// TIA Portal V20 export
FUNCTION "CollectAlarms" : Void   // FC35, LAD
TITLE = U1Em5_CathodeMainPnP
// stored: Namespace Unit1.Em5, SetENOAutomatically false
   VAR_INPUT
      resetAlarms : Bool;
      disableAlarms : Bool;
   END_VAR
   VAR_OUTPUT
      commandsToUnit : "LUC_typeStateCommands";   // Feedback to the unit
   END_VAR
   VAR CONSTANT
      DelayTime : Time := T#300ms;
      NoDelayTime : Time;
   END_VAR
BEGIN

REGION Network 1: Reset Alarms
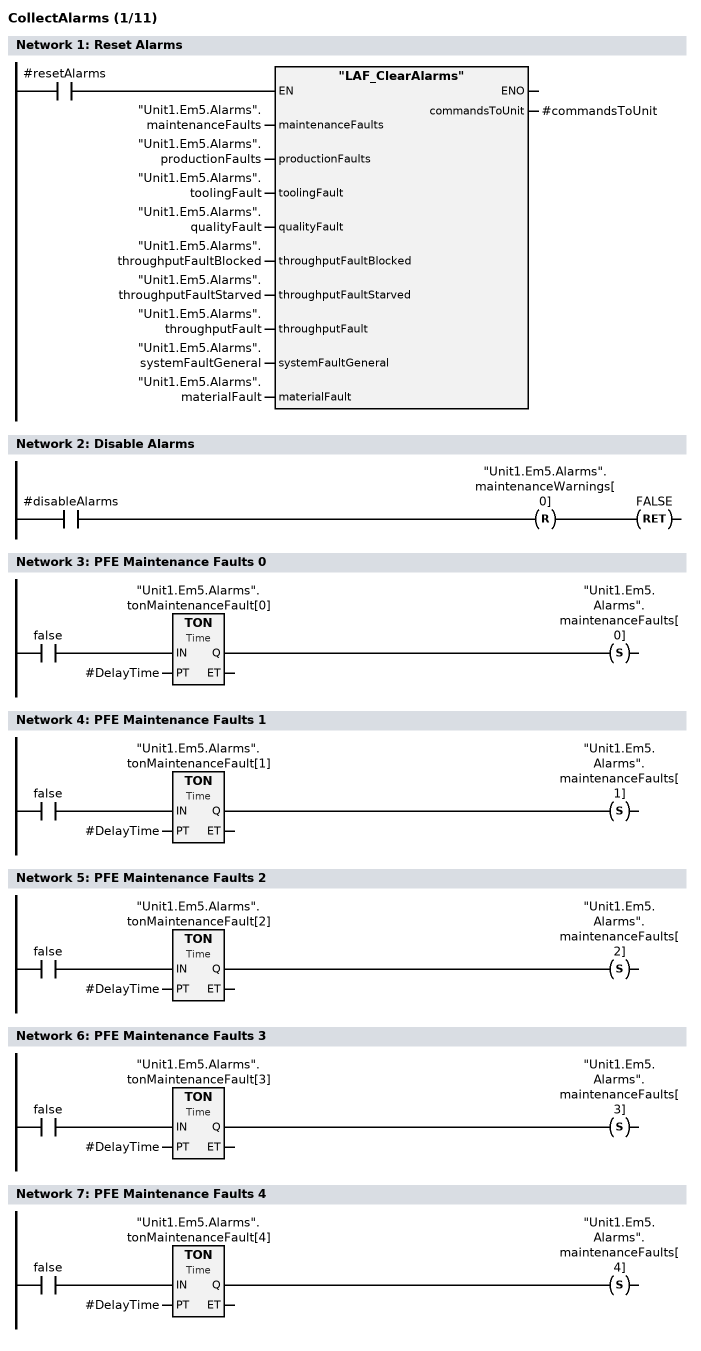
   RUNG wire#powerrail
      Contact( #resetAlarms )
      "LAF_ClearAlarms"(maintenanceFaults := "Unit1.Em5.Alarms".maintenanceFaults, productionFaults := "Unit1.Em5.Alarms".productionFaults, toolingFault := "Unit1.Em5.Alarms".toolingFault, qualityFault := "Unit1.Em5.Alarms".qualityFault, throughputFaultBlocked := "Unit1.Em5.Alarms".throughputFaultBlocked, throughputFaultStarved := "Unit1.Em5.Alarms".throughputFaultStarved, throughputFault := "Unit1.Em5.Alarms".throughputFault, systemFaultGeneral := "Unit1.Em5.Alarms".systemFaultGeneral, materialFault := "Unit1.Em5.Alarms".materialFault, commandsToUnit => #commandsToUnit)
   END_RUNG
   // the same network as SCL:
   IF #resetAlarms THEN
       "LAF_ClearAlarms"(maintenanceFaults := "Unit1.Em5.Alarms".maintenanceFaults,
                         productionFaults := "Unit1.Em5.Alarms".productionFaults,
                         toolingFault := "Unit1.Em5.Alarms".toolingFault,
                         qualityFault := "Unit1.Em5.Alarms".qualityFault,
                         throughputFaultBlocked := "Unit1.Em5.Alarms".throughputFaultBlocked,
                         throughputFaultStarved := "Unit1.Em5.Alarms".throughputFaultStarved,
                         throughputFault := "Unit1.Em5.Alarms".throughputFault,
                         systemFaultGeneral := "Unit1.Em5.Alarms".systemFaultGeneral,
                         materialFault := "Unit1.Em5.Alarms".materialFault,
                         commandsToUnit => #commandsToUnit);
   END_IF;
END_REGION

REGION Network 2: Disable Alarms
   RUNG wire#powerrail
      Contact( #disableAlarms )
      R_Coil( "Unit1.Em5.Alarms".maintenanceWarnings[0] )
      ReturnCoil( FALSE )
   END_RUNG
   // the same network as SCL:
   IF #disableAlarms THEN
       "Unit1.Em5.Alarms".maintenanceWarnings[0] := FALSE;
       ENO := FALSE;
       RETURN;
   END_IF;
END_REGION

REGION Network 3: PFE Maintenance Faults 0
   RUNG wire#powerrail
      Contact( false )
      { S7_Templates := "time_type := Time" } "Unit1.Em5.Alarms".tonMaintenanceFault[0].TON(pt := #DelayTime, et =>)
      S_Coil( "Unit1.Em5.Alarms".maintenanceFaults[0] )
   END_RUNG
   // the same network as SCL:
   "Unit1.Em5.Alarms".tonMaintenanceFault[0].TON(IN := false, PT := #DelayTime);
   IF "Unit1.Em5.Alarms".tonMaintenanceFault[0].Q THEN
       "Unit1.Em5.Alarms".maintenanceFaults[0] := TRUE;
   END_IF;
END_REGION

REGION Network 4: PFE Maintenance Faults 1
   RUNG wire#powerrail
      Contact( false )
      { S7_Templates := "time_type := Time" } "Unit1.Em5.Alarms".tonMaintenanceFault[1].TON(pt := #DelayTime, et =>)
      S_Coil( "Unit1.Em5.Alarms".maintenanceFaults[1] )
   END_RUNG
   // the same network as SCL:
   "Unit1.Em5.Alarms".tonMaintenanceFault[1].TON(IN := false, PT := #DelayTime);
   IF "Unit1.Em5.Alarms".tonMaintenanceFault[1].Q THEN
       "Unit1.Em5.Alarms".maintenanceFaults[1] := TRUE;
   END_IF;
END_REGION

REGION Network 5: PFE Maintenance Faults 2
   RUNG wire#powerrail
      Contact( false )
      { S7_Templates := "time_type := Time" } "Unit1.Em5.Alarms".tonMaintenanceFault[2].TON(pt := #DelayTime, et =>)
      S_Coil( "Unit1.Em5.Alarms".maintenanceFaults[2] )
   END_RUNG
   // the same network as SCL:
   "Unit1.Em5.Alarms".tonMaintenanceFault[2].TON(IN := false, PT := #DelayTime);
   IF "Unit1.Em5.Alarms".tonMaintenanceFault[2].Q THEN
       "Unit1.Em5.Alarms".maintenanceFaults[2] := TRUE;
   END_IF;
END_REGION

REGION Network 6: PFE Maintenance Faults 3
   RUNG wire#powerrail
      Contact( false )
      { S7_Templates := "time_type := Time" } "Unit1.Em5.Alarms".tonMaintenanceFault[3].TON(pt := #DelayTime, et =>)
      S_Coil( "Unit1.Em5.Alarms".maintenanceFaults[3] )
   END_RUNG
   // the same network as SCL:
   "Unit1.Em5.Alarms".tonMaintenanceFault[3].TON(IN := false, PT := #DelayTime);
   IF "Unit1.Em5.Alarms".tonMaintenanceFault[3].Q THEN
       "Unit1.Em5.Alarms".maintenanceFaults[3] := TRUE;
   END_IF;
END_REGION

REGION Network 7: PFE Maintenance Faults 4
   RUNG wire#powerrail
      Contact( false )
      { S7_Templates := "time_type := Time" } "Unit1.Em5.Alarms".tonMaintenanceFault[4].TON(pt := #DelayTime, et =>)
      S_Coil( "Unit1.Em5.Alarms".maintenanceFaults[4] )
   END_RUNG
   // the same network as SCL:
   "Unit1.Em5.Alarms".tonMaintenanceFault[4].TON(IN := false, PT := #DelayTime);
   IF "Unit1.Em5.Alarms".tonMaintenanceFault[4].Q THEN
       "Unit1.Em5.Alarms".maintenanceFaults[4] := TRUE;
   END_IF;
END_REGION

REGION Network 8: PFE Maintenance Faults 5
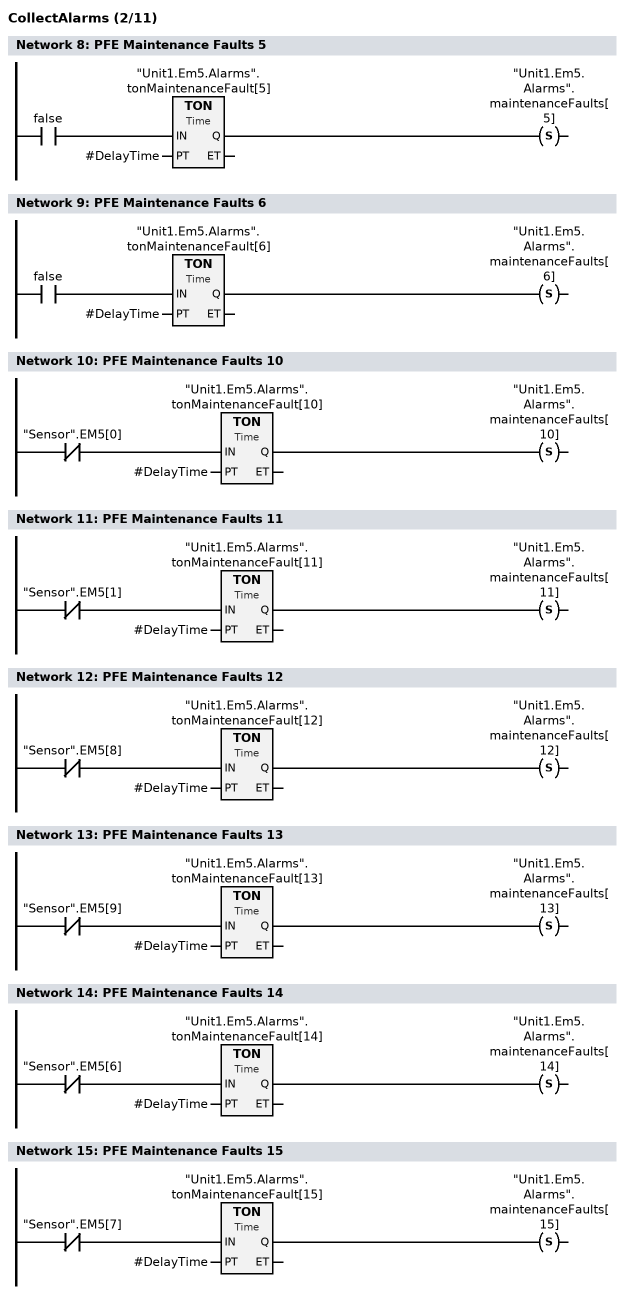
   RUNG wire#powerrail
      Contact( false )
      { S7_Templates := "time_type := Time" } "Unit1.Em5.Alarms".tonMaintenanceFault[5].TON(pt := #DelayTime, et =>)
      S_Coil( "Unit1.Em5.Alarms".maintenanceFaults[5] )
   END_RUNG
   // the same network as SCL:
   "Unit1.Em5.Alarms".tonMaintenanceFault[5].TON(IN := false, PT := #DelayTime);
   IF "Unit1.Em5.Alarms".tonMaintenanceFault[5].Q THEN
       "Unit1.Em5.Alarms".maintenanceFaults[5] := TRUE;
   END_IF;
END_REGION

REGION Network 9: PFE Maintenance Faults 6
   RUNG wire#powerrail
      Contact( false )
      { S7_Templates := "time_type := Time" } "Unit1.Em5.Alarms".tonMaintenanceFault[6].TON(pt := #DelayTime, et =>)
      S_Coil( "Unit1.Em5.Alarms".maintenanceFaults[6] )
   END_RUNG
   // the same network as SCL:
   "Unit1.Em5.Alarms".tonMaintenanceFault[6].TON(IN := false, PT := #DelayTime);
   IF "Unit1.Em5.Alarms".tonMaintenanceFault[6].Q THEN
       "Unit1.Em5.Alarms".maintenanceFaults[6] := TRUE;
   END_IF;
END_REGION

REGION Network 10: PFE Maintenance Faults 10
   RUNG wire#powerrail
      I_Contact( "Sensor".EM5[0] )
      { S7_Templates := "time_type := Time" } "Unit1.Em5.Alarms".tonMaintenanceFault[10].TON(pt := #DelayTime, et =>)
      S_Coil( "Unit1.Em5.Alarms".maintenanceFaults[10] )
   END_RUNG
   // the same network as SCL:
   "Unit1.Em5.Alarms".tonMaintenanceFault[10].TON(IN := NOT "Sensor".EM5[0], PT := #DelayTime);
   IF "Unit1.Em5.Alarms".tonMaintenanceFault[10].Q THEN
       "Unit1.Em5.Alarms".maintenanceFaults[10] := TRUE;
   END_IF;
END_REGION

REGION Network 11: PFE Maintenance Faults 11
   RUNG wire#powerrail
      I_Contact( "Sensor".EM5[1] )
      { S7_Templates := "time_type := Time" } "Unit1.Em5.Alarms".tonMaintenanceFault[11].TON(pt := #DelayTime, et =>)
      S_Coil( "Unit1.Em5.Alarms".maintenanceFaults[11] )
   END_RUNG
   // the same network as SCL:
   "Unit1.Em5.Alarms".tonMaintenanceFault[11].TON(IN := NOT "Sensor".EM5[1], PT := #DelayTime);
   IF "Unit1.Em5.Alarms".tonMaintenanceFault[11].Q THEN
       "Unit1.Em5.Alarms".maintenanceFaults[11] := TRUE;
   END_IF;
END_REGION

REGION Network 12: PFE Maintenance Faults 12
   RUNG wire#powerrail
      I_Contact( "Sensor".EM5[8] )
      { S7_Templates := "time_type := Time" } "Unit1.Em5.Alarms".tonMaintenanceFault[12].TON(pt := #DelayTime, et =>)
      S_Coil( "Unit1.Em5.Alarms".maintenanceFaults[12] )
   END_RUNG
   // the same network as SCL:
   "Unit1.Em5.Alarms".tonMaintenanceFault[12].TON(IN := NOT "Sensor".EM5[8], PT := #DelayTime);
   IF "Unit1.Em5.Alarms".tonMaintenanceFault[12].Q THEN
       "Unit1.Em5.Alarms".maintenanceFaults[12] := TRUE;
   END_IF;
END_REGION

REGION Network 13: PFE Maintenance Faults 13
   RUNG wire#powerrail
      I_Contact( "Sensor".EM5[9] )
      { S7_Templates := "time_type := Time" } "Unit1.Em5.Alarms".tonMaintenanceFault[13].TON(pt := #DelayTime, et =>)
      S_Coil( "Unit1.Em5.Alarms".maintenanceFaults[13] )
   END_RUNG
   // the same network as SCL:
   "Unit1.Em5.Alarms".tonMaintenanceFault[13].TON(IN := NOT "Sensor".EM5[9], PT := #DelayTime);
   IF "Unit1.Em5.Alarms".tonMaintenanceFault[13].Q THEN
       "Unit1.Em5.Alarms".maintenanceFaults[13] := TRUE;
   END_IF;
END_REGION

REGION Network 14: PFE Maintenance Faults 14
   RUNG wire#powerrail
      I_Contact( "Sensor".EM5[6] )
      { S7_Templates := "time_type := Time" } "Unit1.Em5.Alarms".tonMaintenanceFault[14].TON(pt := #DelayTime, et =>)
      S_Coil( "Unit1.Em5.Alarms".maintenanceFaults[14] )
   END_RUNG
   // the same network as SCL:
   "Unit1.Em5.Alarms".tonMaintenanceFault[14].TON(IN := NOT "Sensor".EM5[6], PT := #DelayTime);
   IF "Unit1.Em5.Alarms".tonMaintenanceFault[14].Q THEN
       "Unit1.Em5.Alarms".maintenanceFaults[14] := TRUE;
   END_IF;
END_REGION

REGION Network 15: PFE Maintenance Faults 15
   RUNG wire#powerrail
      I_Contact( "Sensor".EM5[7] )
      { S7_Templates := "time_type := Time" } "Unit1.Em5.Alarms".tonMaintenanceFault[15].TON(pt := #DelayTime, et =>)
      S_Coil( "Unit1.Em5.Alarms".maintenanceFaults[15] )
   END_RUNG
   // the same network as SCL:
   "Unit1.Em5.Alarms".tonMaintenanceFault[15].TON(IN := NOT "Sensor".EM5[7], PT := #DelayTime);
   IF "Unit1.Em5.Alarms".tonMaintenanceFault[15].Q THEN
       "Unit1.Em5.Alarms".maintenanceFaults[15] := TRUE;
   END_IF;
END_REGION

REGION Network 16: PFE Maintenance Faults 16
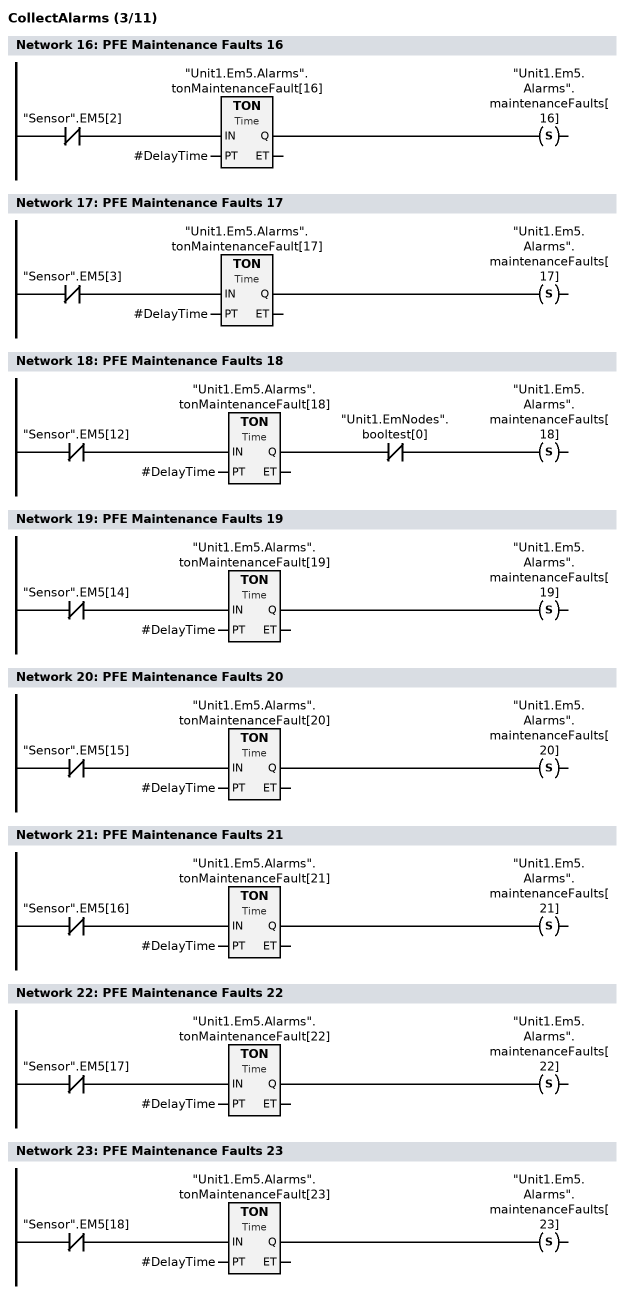
   RUNG wire#powerrail
      I_Contact( "Sensor".EM5[2] )
      { S7_Templates := "time_type := Time" } "Unit1.Em5.Alarms".tonMaintenanceFault[16].TON(pt := #DelayTime, et =>)
      S_Coil( "Unit1.Em5.Alarms".maintenanceFaults[16] )
   END_RUNG
   // the same network as SCL:
   "Unit1.Em5.Alarms".tonMaintenanceFault[16].TON(IN := NOT "Sensor".EM5[2], PT := #DelayTime);
   IF "Unit1.Em5.Alarms".tonMaintenanceFault[16].Q THEN
       "Unit1.Em5.Alarms".maintenanceFaults[16] := TRUE;
   END_IF;
END_REGION

REGION Network 17: PFE Maintenance Faults 17
   RUNG wire#powerrail
      I_Contact( "Sensor".EM5[3] )
      { S7_Templates := "time_type := Time" } "Unit1.Em5.Alarms".tonMaintenanceFault[17].TON(pt := #DelayTime, et =>)
      S_Coil( "Unit1.Em5.Alarms".maintenanceFaults[17] )
   END_RUNG
   // the same network as SCL:
   "Unit1.Em5.Alarms".tonMaintenanceFault[17].TON(IN := NOT "Sensor".EM5[3], PT := #DelayTime);
   IF "Unit1.Em5.Alarms".tonMaintenanceFault[17].Q THEN
       "Unit1.Em5.Alarms".maintenanceFaults[17] := TRUE;
   END_IF;
END_REGION

REGION Network 18: PFE Maintenance Faults 18
   RUNG wire#powerrail
      I_Contact( "Sensor".EM5[12] )
      { S7_Templates := "time_type := Time" } "Unit1.Em5.Alarms".tonMaintenanceFault[18].TON(pt := #DelayTime, et =>)
      I_Contact( "Unit1.EmNodes".booltest[0] )
      S_Coil( "Unit1.Em5.Alarms".maintenanceFaults[18] )
   END_RUNG
   // the same network as SCL:
   "Unit1.Em5.Alarms".tonMaintenanceFault[18].TON(IN := NOT "Sensor".EM5[12], PT := #DelayTime);
   IF "Unit1.Em5.Alarms".tonMaintenanceFault[18].Q AND NOT "Unit1.EmNodes".booltest[0] THEN
       "Unit1.Em5.Alarms".maintenanceFaults[18] := TRUE;
   END_IF;
END_REGION

REGION Network 19: PFE Maintenance Faults 19
   RUNG wire#powerrail
      I_Contact( "Sensor".EM5[14] )
      { S7_Templates := "time_type := Time" } "Unit1.Em5.Alarms".tonMaintenanceFault[19].TON(pt := #DelayTime, et =>)
      S_Coil( "Unit1.Em5.Alarms".maintenanceFaults[19] )
   END_RUNG
   // the same network as SCL:
   "Unit1.Em5.Alarms".tonMaintenanceFault[19].TON(IN := NOT "Sensor".EM5[14], PT := #DelayTime);
   IF "Unit1.Em5.Alarms".tonMaintenanceFault[19].Q THEN
       "Unit1.Em5.Alarms".maintenanceFaults[19] := TRUE;
   END_IF;
END_REGION

REGION Network 20: PFE Maintenance Faults 20
   RUNG wire#powerrail
      I_Contact( "Sensor".EM5[15] )
      { S7_Templates := "time_type := Time" } "Unit1.Em5.Alarms".tonMaintenanceFault[20].TON(pt := #DelayTime, et =>)
      S_Coil( "Unit1.Em5.Alarms".maintenanceFaults[20] )
   END_RUNG
   // the same network as SCL:
   "Unit1.Em5.Alarms".tonMaintenanceFault[20].TON(IN := NOT "Sensor".EM5[15], PT := #DelayTime);
   IF "Unit1.Em5.Alarms".tonMaintenanceFault[20].Q THEN
       "Unit1.Em5.Alarms".maintenanceFaults[20] := TRUE;
   END_IF;
END_REGION

REGION Network 21: PFE Maintenance Faults 21
   RUNG wire#powerrail
      I_Contact( "Sensor".EM5[16] )
      { S7_Templates := "time_type := Time" } "Unit1.Em5.Alarms".tonMaintenanceFault[21].TON(pt := #DelayTime, et =>)
      S_Coil( "Unit1.Em5.Alarms".maintenanceFaults[21] )
   END_RUNG
   // the same network as SCL:
   "Unit1.Em5.Alarms".tonMaintenanceFault[21].TON(IN := NOT "Sensor".EM5[16], PT := #DelayTime);
   IF "Unit1.Em5.Alarms".tonMaintenanceFault[21].Q THEN
       "Unit1.Em5.Alarms".maintenanceFaults[21] := TRUE;
   END_IF;
END_REGION

REGION Network 22: PFE Maintenance Faults 22
   RUNG wire#powerrail
      I_Contact( "Sensor".EM5[17] )
      { S7_Templates := "time_type := Time" } "Unit1.Em5.Alarms".tonMaintenanceFault[22].TON(pt := #DelayTime, et =>)
      S_Coil( "Unit1.Em5.Alarms".maintenanceFaults[22] )
   END_RUNG
   // the same network as SCL:
   "Unit1.Em5.Alarms".tonMaintenanceFault[22].TON(IN := NOT "Sensor".EM5[17], PT := #DelayTime);
   IF "Unit1.Em5.Alarms".tonMaintenanceFault[22].Q THEN
       "Unit1.Em5.Alarms".maintenanceFaults[22] := TRUE;
   END_IF;
END_REGION

REGION Network 23: PFE Maintenance Faults 23
   RUNG wire#powerrail
      I_Contact( "Sensor".EM5[18] )
      { S7_Templates := "time_type := Time" } "Unit1.Em5.Alarms".tonMaintenanceFault[23].TON(pt := #DelayTime, et =>)
      S_Coil( "Unit1.Em5.Alarms".maintenanceFaults[23] )
   END_RUNG
   // the same network as SCL:
   "Unit1.Em5.Alarms".tonMaintenanceFault[23].TON(IN := NOT "Sensor".EM5[18], PT := #DelayTime);
   IF "Unit1.Em5.Alarms".tonMaintenanceFault[23].Q THEN
       "Unit1.Em5.Alarms".maintenanceFaults[23] := TRUE;
   END_IF;
END_REGION

REGION Network 24: PFE Maintenance Faults 24
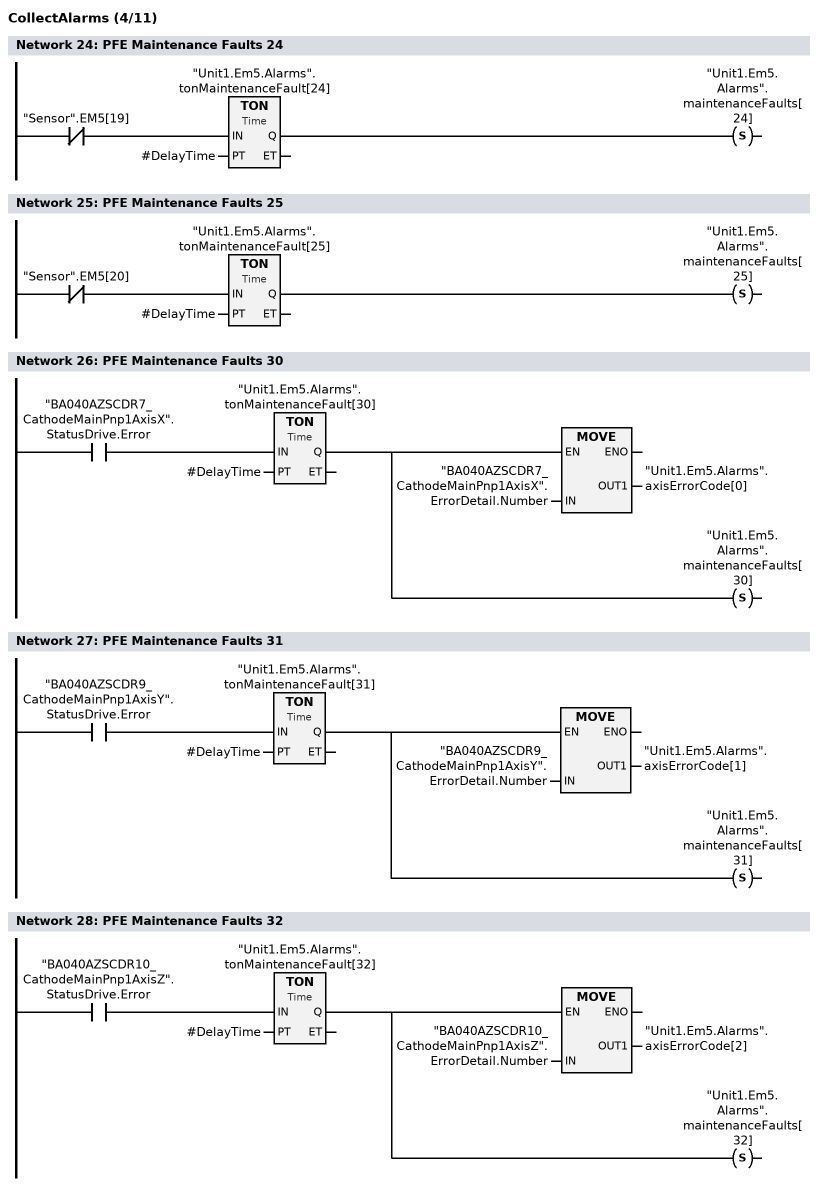
   RUNG wire#powerrail
      I_Contact( "Sensor".EM5[19] )
      { S7_Templates := "time_type := Time" } "Unit1.Em5.Alarms".tonMaintenanceFault[24].TON(pt := #DelayTime, et =>)
      S_Coil( "Unit1.Em5.Alarms".maintenanceFaults[24] )
   END_RUNG
   // the same network as SCL:
   "Unit1.Em5.Alarms".tonMaintenanceFault[24].TON(IN := NOT "Sensor".EM5[19], PT := #DelayTime);
   IF "Unit1.Em5.Alarms".tonMaintenanceFault[24].Q THEN
       "Unit1.Em5.Alarms".maintenanceFaults[24] := TRUE;
   END_IF;
END_REGION

REGION Network 25: PFE Maintenance Faults 25
   RUNG wire#powerrail
      I_Contact( "Sensor".EM5[20] )
      { S7_Templates := "time_type := Time" } "Unit1.Em5.Alarms".tonMaintenanceFault[25].TON(pt := #DelayTime, et =>)
      S_Coil( "Unit1.Em5.Alarms".maintenanceFaults[25] )
   END_RUNG
   // the same network as SCL:
   "Unit1.Em5.Alarms".tonMaintenanceFault[25].TON(IN := NOT "Sensor".EM5[20], PT := #DelayTime);
   IF "Unit1.Em5.Alarms".tonMaintenanceFault[25].Q THEN
       "Unit1.Em5.Alarms".maintenanceFaults[25] := TRUE;
   END_IF;
END_REGION

REGION Network 26: PFE Maintenance Faults 30
   RUNG wire#powerrail
      Contact( "BA040AZSCDR7_CathodeMainPnp1AxisX".StatusDrive.Error )
      { S7_Templates := "time_type := Time" } "Unit1.Em5.Alarms".tonMaintenanceFault[30].TON(pt := #DelayTime, et =>)
      wire#w1
      Move(in := "BA040AZSCDR7_CathodeMainPnp1AxisX".ErrorDetail.Number, out1 => "Unit1.Em5.Alarms".axisErrorCode[0])
   END_RUNG
   RUNG wire#w1
      S_Coil( "Unit1.Em5.Alarms".maintenanceFaults[30] )
   END_RUNG
   // the same network as SCL:
   "Unit1.Em5.Alarms".tonMaintenanceFault[30].TON(IN := "BA040AZSCDR7_CathodeMainPnp1AxisX".StatusDrive.Error,
                           PT := #DelayTime);
   IF "Unit1.Em5.Alarms".tonMaintenanceFault[30].Q THEN
       "Unit1.Em5.Alarms".axisErrorCode[0] := "BA040AZSCDR7_CathodeMainPnp1AxisX".ErrorDetail.Number;
       "Unit1.Em5.Alarms".maintenanceFaults[30] := TRUE;
   END_IF;
END_REGION

REGION Network 27: PFE Maintenance Faults 31
   RUNG wire#powerrail
      Contact( "BA040AZSCDR9_CathodeMainPnp1AxisY".StatusDrive.Error )
      { S7_Templates := "time_type := Time" } "Unit1.Em5.Alarms".tonMaintenanceFault[31].TON(pt := #DelayTime, et =>)
      wire#w1
      Move(in := "BA040AZSCDR9_CathodeMainPnp1AxisY".ErrorDetail.Number, out1 => "Unit1.Em5.Alarms".axisErrorCode[1])
   END_RUNG
   RUNG wire#w1
      S_Coil( "Unit1.Em5.Alarms".maintenanceFaults[31] )
   END_RUNG
   // the same network as SCL:
   "Unit1.Em5.Alarms".tonMaintenanceFault[31].TON(IN := "BA040AZSCDR9_CathodeMainPnp1AxisY".StatusDrive.Error,
                           PT := #DelayTime);
   IF "Unit1.Em5.Alarms".tonMaintenanceFault[31].Q THEN
       "Unit1.Em5.Alarms".axisErrorCode[1] := "BA040AZSCDR9_CathodeMainPnp1AxisY".ErrorDetail.Number;
       "Unit1.Em5.Alarms".maintenanceFaults[31] := TRUE;
   END_IF;
END_REGION

REGION Network 28: PFE Maintenance Faults 32
   RUNG wire#powerrail
      Contact( "BA040AZSCDR10_CathodeMainPnp1AxisZ".StatusDrive.Error )
      { S7_Templates := "time_type := Time" } "Unit1.Em5.Alarms".tonMaintenanceFault[32].TON(pt := #DelayTime, et =>)
      wire#w1
      Move(in := "BA040AZSCDR10_CathodeMainPnp1AxisZ".ErrorDetail.Number, out1 => "Unit1.Em5.Alarms".axisErrorCode[2])
   END_RUNG
   RUNG wire#w1
      S_Coil( "Unit1.Em5.Alarms".maintenanceFaults[32] )
   END_RUNG
   // the same network as SCL:
   "Unit1.Em5.Alarms".tonMaintenanceFault[32].TON(IN := "BA040AZSCDR10_CathodeMainPnp1AxisZ".StatusDrive.Error,
                           PT := #DelayTime);
   IF "Unit1.Em5.Alarms".tonMaintenanceFault[32].Q THEN
       "Unit1.Em5.Alarms".axisErrorCode[2] := "BA040AZSCDR10_CathodeMainPnp1AxisZ".ErrorDetail.Number;
       "Unit1.Em5.Alarms".maintenanceFaults[32] := TRUE;
   END_IF;
END_REGION

REGION Network 29: PFE Maintenance Faults 33
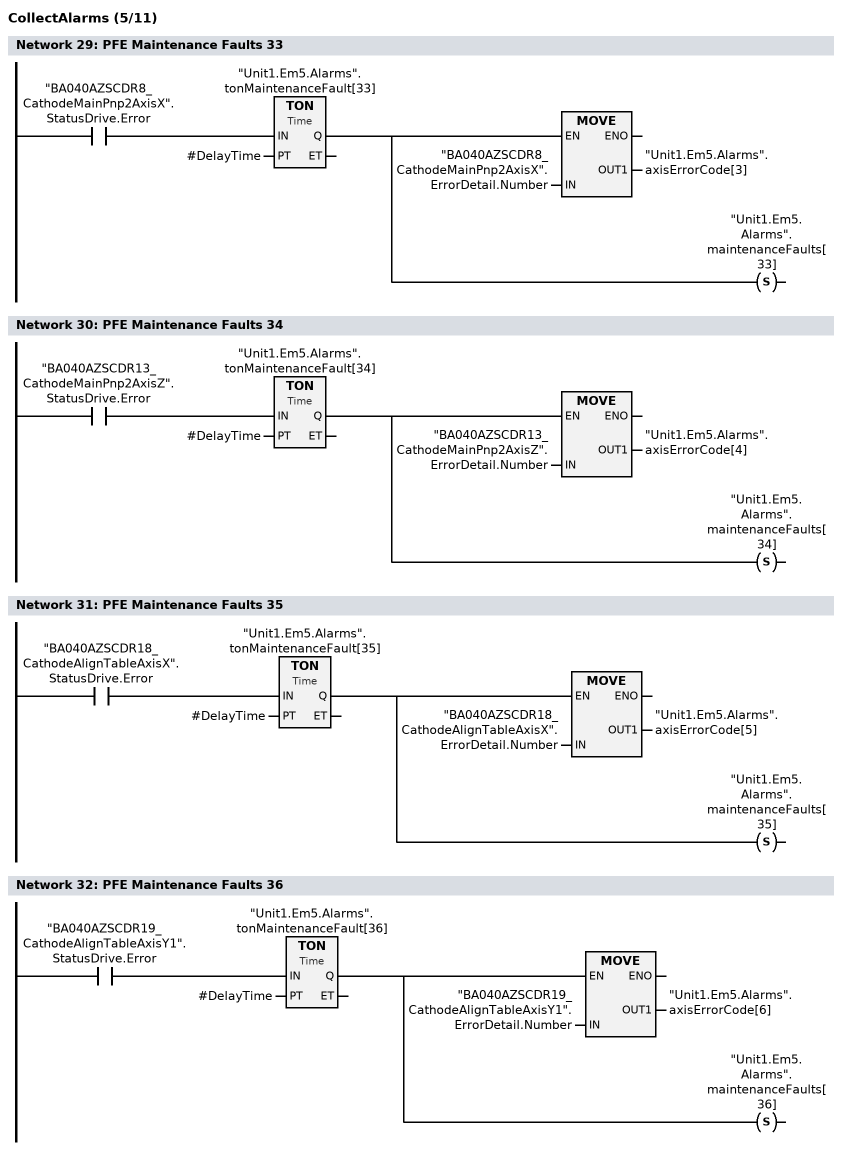
   RUNG wire#powerrail
      Contact( "BA040AZSCDR8_CathodeMainPnp2AxisX".StatusDrive.Error )
      { S7_Templates := "time_type := Time" } "Unit1.Em5.Alarms".tonMaintenanceFault[33].TON(pt := #DelayTime, et =>)
      wire#w1
      Move(in := "BA040AZSCDR8_CathodeMainPnp2AxisX".ErrorDetail.Number, out1 => "Unit1.Em5.Alarms".axisErrorCode[3])
   END_RUNG
   RUNG wire#w1
      S_Coil( "Unit1.Em5.Alarms".maintenanceFaults[33] )
   END_RUNG
   // the same network as SCL:
   "Unit1.Em5.Alarms".tonMaintenanceFault[33].TON(IN := "BA040AZSCDR8_CathodeMainPnp2AxisX".StatusDrive.Error,
                           PT := #DelayTime);
   IF "Unit1.Em5.Alarms".tonMaintenanceFault[33].Q THEN
       "Unit1.Em5.Alarms".axisErrorCode[3] := "BA040AZSCDR8_CathodeMainPnp2AxisX".ErrorDetail.Number;
       "Unit1.Em5.Alarms".maintenanceFaults[33] := TRUE;
   END_IF;
END_REGION

REGION Network 30: PFE Maintenance Faults 34
   RUNG wire#powerrail
      Contact( "BA040AZSCDR13_CathodeMainPnp2AxisZ".StatusDrive.Error )
      { S7_Templates := "time_type := Time" } "Unit1.Em5.Alarms".tonMaintenanceFault[34].TON(pt := #DelayTime, et =>)
      wire#w1
      Move(in := "BA040AZSCDR13_CathodeMainPnp2AxisZ".ErrorDetail.Number, out1 => "Unit1.Em5.Alarms".axisErrorCode[4])
   END_RUNG
   RUNG wire#w1
      S_Coil( "Unit1.Em5.Alarms".maintenanceFaults[34] )
   END_RUNG
   // the same network as SCL:
   "Unit1.Em5.Alarms".tonMaintenanceFault[34].TON(IN := "BA040AZSCDR13_CathodeMainPnp2AxisZ".StatusDrive.Error,
                           PT := #DelayTime);
   IF "Unit1.Em5.Alarms".tonMaintenanceFault[34].Q THEN
       "Unit1.Em5.Alarms".axisErrorCode[4] := "BA040AZSCDR13_CathodeMainPnp2AxisZ".ErrorDetail.Number;
       "Unit1.Em5.Alarms".maintenanceFaults[34] := TRUE;
   END_IF;
END_REGION

REGION Network 31: PFE Maintenance Faults 35
   RUNG wire#powerrail
      Contact( "BA040AZSCDR18_CathodeAlignTableAxisX".StatusDrive.Error )
      { S7_Templates := "time_type := Time" } "Unit1.Em5.Alarms".tonMaintenanceFault[35].TON(pt := #DelayTime, et =>)
      wire#w1
      Move(in := "BA040AZSCDR18_CathodeAlignTableAxisX".ErrorDetail.Number, out1 => "Unit1.Em5.Alarms".axisErrorCode[5])
   END_RUNG
   RUNG wire#w1
      S_Coil( "Unit1.Em5.Alarms".maintenanceFaults[35] )
   END_RUNG
   // the same network as SCL:
   "Unit1.Em5.Alarms".tonMaintenanceFault[35].TON(IN := "BA040AZSCDR18_CathodeAlignTableAxisX".StatusDrive.Error,
                           PT := #DelayTime);
   IF "Unit1.Em5.Alarms".tonMaintenanceFault[35].Q THEN
       "Unit1.Em5.Alarms".axisErrorCode[5] := "BA040AZSCDR18_CathodeAlignTableAxisX".ErrorDetail.Number;
       "Unit1.Em5.Alarms".maintenanceFaults[35] := TRUE;
   END_IF;
END_REGION

REGION Network 32: PFE Maintenance Faults 36
   RUNG wire#powerrail
      Contact( "BA040AZSCDR19_CathodeAlignTableAxisY1".StatusDrive.Error )
      { S7_Templates := "time_type := Time" } "Unit1.Em5.Alarms".tonMaintenanceFault[36].TON(pt := #DelayTime, et =>)
      wire#w1
      Move(in := "BA040AZSCDR19_CathodeAlignTableAxisY1".ErrorDetail.Number, out1 => "Unit1.Em5.Alarms".axisErrorCode[6])
   END_RUNG
   RUNG wire#w1
      S_Coil( "Unit1.Em5.Alarms".maintenanceFaults[36] )
   END_RUNG
   // the same network as SCL:
   "Unit1.Em5.Alarms".tonMaintenanceFault[36].TON(IN := "BA040AZSCDR19_CathodeAlignTableAxisY1".StatusDrive.Error,
                           PT := #DelayTime);
   IF "Unit1.Em5.Alarms".tonMaintenanceFault[36].Q THEN
       "Unit1.Em5.Alarms".axisErrorCode[6] := "BA040AZSCDR19_CathodeAlignTableAxisY1".ErrorDetail.Number;
       "Unit1.Em5.Alarms".maintenanceFaults[36] := TRUE;
   END_IF;
END_REGION

REGION Network 33: PFE Maintenance Faults 37
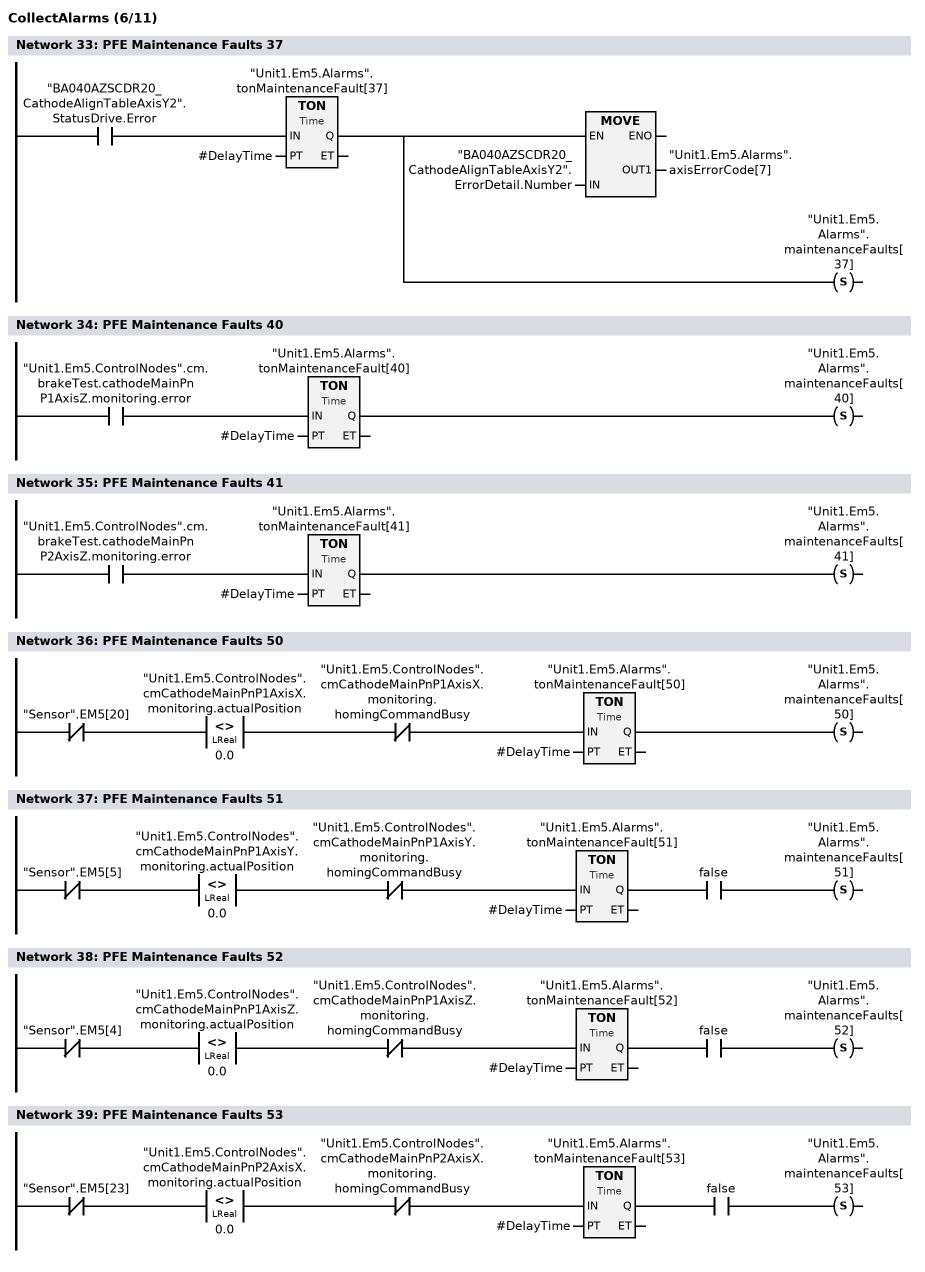
   RUNG wire#powerrail
      Contact( "BA040AZSCDR20_CathodeAlignTableAxisY2".StatusDrive.Error )
      { S7_Templates := "time_type := Time" } "Unit1.Em5.Alarms".tonMaintenanceFault[37].TON(pt := #DelayTime, et =>)
      wire#w1
      Move(in := "BA040AZSCDR20_CathodeAlignTableAxisY2".ErrorDetail.Number, out1 => "Unit1.Em5.Alarms".axisErrorCode[7])
   END_RUNG
   RUNG wire#w1
      S_Coil( "Unit1.Em5.Alarms".maintenanceFaults[37] )
   END_RUNG
   // the same network as SCL:
   "Unit1.Em5.Alarms".tonMaintenanceFault[37].TON(IN := "BA040AZSCDR20_CathodeAlignTableAxisY2".StatusDrive.Error,
                           PT := #DelayTime);
   IF "Unit1.Em5.Alarms".tonMaintenanceFault[37].Q THEN
       "Unit1.Em5.Alarms".axisErrorCode[7] := "BA040AZSCDR20_CathodeAlignTableAxisY2".ErrorDetail.Number;
       "Unit1.Em5.Alarms".maintenanceFaults[37] := TRUE;
   END_IF;
END_REGION

REGION Network 34: PFE Maintenance Faults 40
   RUNG wire#powerrail
      Contact( "Unit1.Em5.ControlNodes".cm.brakeTest.cathodeMainPnP1AxisZ.monitoring.error )
      { S7_Templates := "time_type := Time" } "Unit1.Em5.Alarms".tonMaintenanceFault[40].TON(pt := #DelayTime, et =>)
      S_Coil( "Unit1.Em5.Alarms".maintenanceFaults[40] )
   END_RUNG
   // the same network as SCL:
   "Unit1.Em5.Alarms".tonMaintenanceFault[40].TON(IN := "Unit1.Em5.ControlNodes".cm.brakeTest.cathodeMainPnP1AxisZ.monitoring.error,
                           PT := #DelayTime);
   IF "Unit1.Em5.Alarms".tonMaintenanceFault[40].Q THEN
       "Unit1.Em5.Alarms".maintenanceFaults[40] := TRUE;
   END_IF;
END_REGION

REGION Network 35: PFE Maintenance Faults 41
   RUNG wire#powerrail
      Contact( "Unit1.Em5.ControlNodes".cm.brakeTest.cathodeMainPnP2AxisZ.monitoring.error )
      { S7_Templates := "time_type := Time" } "Unit1.Em5.Alarms".tonMaintenanceFault[41].TON(pt := #DelayTime, et =>)
      S_Coil( "Unit1.Em5.Alarms".maintenanceFaults[41] )
   END_RUNG
   // the same network as SCL:
   "Unit1.Em5.Alarms".tonMaintenanceFault[41].TON(IN := "Unit1.Em5.ControlNodes".cm.brakeTest.cathodeMainPnP2AxisZ.monitoring.error,
                           PT := #DelayTime);
   IF "Unit1.Em5.Alarms".tonMaintenanceFault[41].Q THEN
       "Unit1.Em5.Alarms".maintenanceFaults[41] := TRUE;
   END_IF;
END_REGION

REGION Network 36: PFE Maintenance Faults 50
   RUNG wire#powerrail
      I_Contact( "Sensor".EM5[20] )
      { S7_Templates := "SrcType := LReal" } NE_Contact(in1 := "Unit1.Em5.ControlNodes".cmCathodeMainPnP1AxisX.monitoring.actualPosition, in2 := 0.0)
      I_Contact( "Unit1.Em5.ControlNodes".cmCathodeMainPnP1AxisX.monitoring.homingCommandBusy )
      { S7_Templates := "time_type := Time" } "Unit1.Em5.Alarms".tonMaintenanceFault[50].TON(pt := #DelayTime, et =>)
      S_Coil( "Unit1.Em5.Alarms".maintenanceFaults[50] )
   END_RUNG
   // the same network as SCL:
   "Unit1.Em5.Alarms".tonMaintenanceFault[50].TON(IN := NOT "Sensor".EM5[20] AND ("Unit1.Em5.ControlNodes".cmCathodeMainPnP1AxisX.monitoring.actualPosition <> 0.0) AND NOT "Unit1.Em5.ControlNodes".cmCathodeMainPnP1AxisX.monitoring.homingCommandBusy,
                           PT := #DelayTime);
   IF "Unit1.Em5.Alarms".tonMaintenanceFault[50].Q THEN
       "Unit1.Em5.Alarms".maintenanceFaults[50] := TRUE;
   END_IF;
END_REGION

REGION Network 37: PFE Maintenance Faults 51
   RUNG wire#powerrail
      I_Contact( "Sensor".EM5[5] )
      { S7_Templates := "SrcType := LReal" } NE_Contact(in1 := "Unit1.Em5.ControlNodes".cmCathodeMainPnP1AxisY.monitoring.actualPosition, in2 := 0.0)
      I_Contact( "Unit1.Em5.ControlNodes".cmCathodeMainPnP1AxisY.monitoring.homingCommandBusy )
      { S7_Templates := "time_type := Time" } "Unit1.Em5.Alarms".tonMaintenanceFault[51].TON(pt := #DelayTime, et =>)
      Contact( false )
      S_Coil( "Unit1.Em5.Alarms".maintenanceFaults[51] )
   END_RUNG
   // the same network as SCL:
   "Unit1.Em5.Alarms".tonMaintenanceFault[51].TON(IN := NOT "Sensor".EM5[5] AND ("Unit1.Em5.ControlNodes".cmCathodeMainPnP1AxisY.monitoring.actualPosition <> 0.0) AND NOT "Unit1.Em5.ControlNodes".cmCathodeMainPnP1AxisY.monitoring.homingCommandBusy,
                           PT := #DelayTime);
   IF "Unit1.Em5.Alarms".tonMaintenanceFault[51].Q AND false THEN
       "Unit1.Em5.Alarms".maintenanceFaults[51] := TRUE;
   END_IF;
END_REGION

REGION Network 38: PFE Maintenance Faults 52
   RUNG wire#powerrail
      I_Contact( "Sensor".EM5[4] )
      { S7_Templates := "SrcType := LReal" } NE_Contact(in1 := "Unit1.Em5.ControlNodes".cmCathodeMainPnP1AxisZ.monitoring.actualPosition, in2 := 0.0)
      I_Contact( "Unit1.Em5.ControlNodes".cmCathodeMainPnP1AxisZ.monitoring.homingCommandBusy )
      { S7_Templates := "time_type := Time" } "Unit1.Em5.Alarms".tonMaintenanceFault[52].TON(pt := #DelayTime, et =>)
      Contact( false )
      S_Coil( "Unit1.Em5.Alarms".maintenanceFaults[52] )
   END_RUNG
   // the same network as SCL:
   "Unit1.Em5.Alarms".tonMaintenanceFault[52].TON(IN := NOT "Sensor".EM5[4] AND ("Unit1.Em5.ControlNodes".cmCathodeMainPnP1AxisZ.monitoring.actualPosition <> 0.0) AND NOT "Unit1.Em5.ControlNodes".cmCathodeMainPnP1AxisZ.monitoring.homingCommandBusy,
                           PT := #DelayTime);
   IF "Unit1.Em5.Alarms".tonMaintenanceFault[52].Q AND false THEN
       "Unit1.Em5.Alarms".maintenanceFaults[52] := TRUE;
   END_IF;
END_REGION

REGION Network 39: PFE Maintenance Faults 53
   RUNG wire#powerrail
      I_Contact( "Sensor".EM5[23] )
      { S7_Templates := "SrcType := LReal" } NE_Contact(in1 := "Unit1.Em5.ControlNodes".cmCathodeMainPnP2AxisX.monitoring.actualPosition, in2 := 0.0)
      I_Contact( "Unit1.Em5.ControlNodes".cmCathodeMainPnP2AxisX.monitoring.homingCommandBusy )
      { S7_Templates := "time_type := Time" } "Unit1.Em5.Alarms".tonMaintenanceFault[53].TON(pt := #DelayTime, et =>)
      Contact( false )
      S_Coil( "Unit1.Em5.Alarms".maintenanceFaults[53] )
   END_RUNG
   // the same network as SCL:
   "Unit1.Em5.Alarms".tonMaintenanceFault[53].TON(IN := NOT "Sensor".EM5[23] AND ("Unit1.Em5.ControlNodes".cmCathodeMainPnP2AxisX.monitoring.actualPosition <> 0.0) AND NOT "Unit1.Em5.ControlNodes".cmCathodeMainPnP2AxisX.monitoring.homingCommandBusy,
                           PT := #DelayTime);
   IF "Unit1.Em5.Alarms".tonMaintenanceFault[53].Q AND false THEN
       "Unit1.Em5.Alarms".maintenanceFaults[53] := TRUE;
   END_IF;
END_REGION

REGION Network 40: PFE Maintenance Faults 54
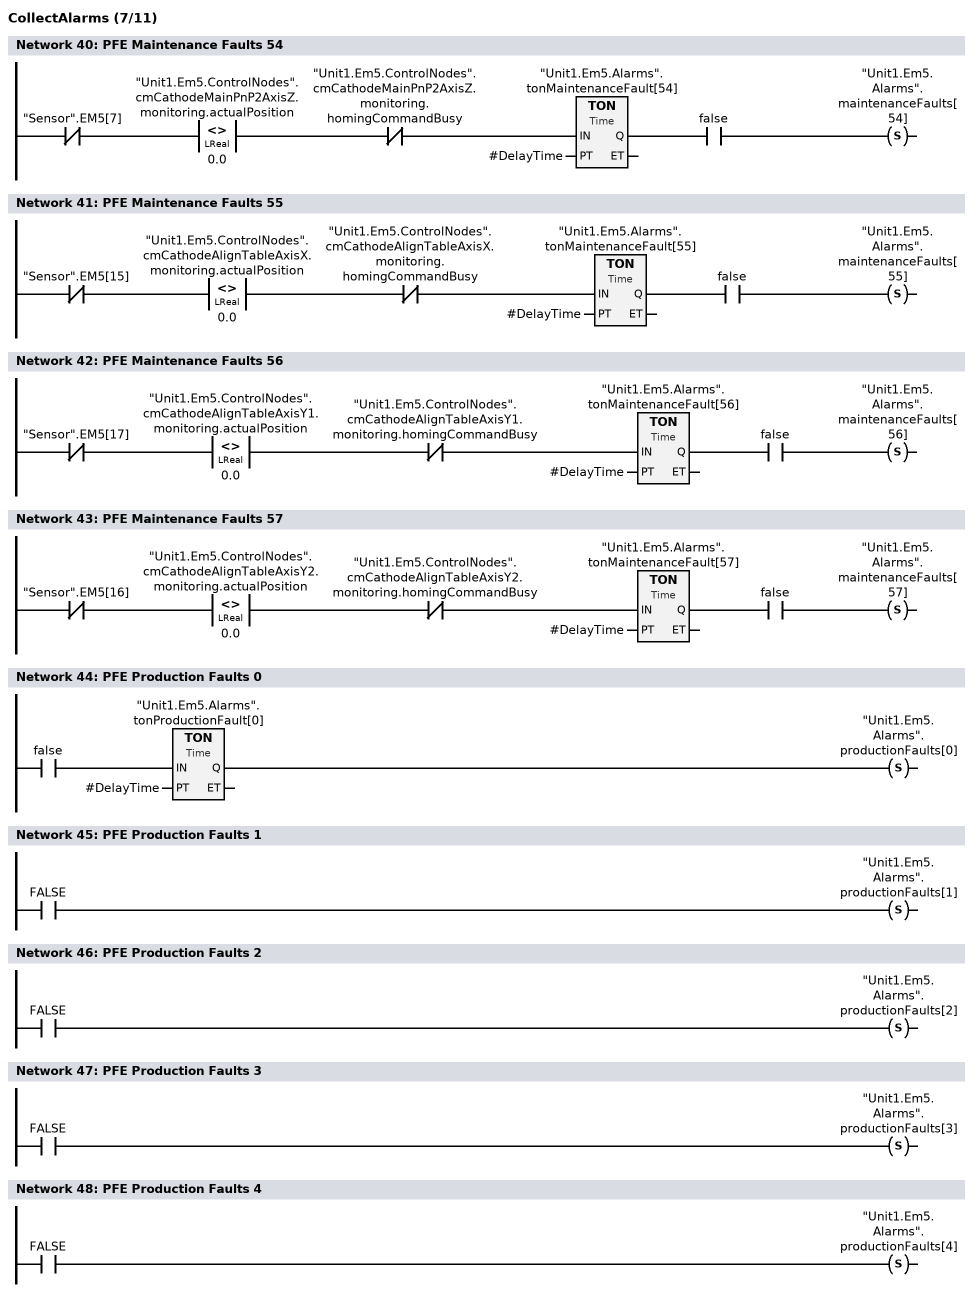
   RUNG wire#powerrail
      I_Contact( "Sensor".EM5[7] )
      { S7_Templates := "SrcType := LReal" } NE_Contact(in1 := "Unit1.Em5.ControlNodes".cmCathodeMainPnP2AxisZ.monitoring.actualPosition, in2 := 0.0)
      I_Contact( "Unit1.Em5.ControlNodes".cmCathodeMainPnP2AxisZ.monitoring.homingCommandBusy )
      { S7_Templates := "time_type := Time" } "Unit1.Em5.Alarms".tonMaintenanceFault[54].TON(pt := #DelayTime, et =>)
      Contact( false )
      S_Coil( "Unit1.Em5.Alarms".maintenanceFaults[54] )
   END_RUNG
   // the same network as SCL:
   "Unit1.Em5.Alarms".tonMaintenanceFault[54].TON(IN := NOT "Sensor".EM5[7] AND ("Unit1.Em5.ControlNodes".cmCathodeMainPnP2AxisZ.monitoring.actualPosition <> 0.0) AND NOT "Unit1.Em5.ControlNodes".cmCathodeMainPnP2AxisZ.monitoring.homingCommandBusy,
                           PT := #DelayTime);
   IF "Unit1.Em5.Alarms".tonMaintenanceFault[54].Q AND false THEN
       "Unit1.Em5.Alarms".maintenanceFaults[54] := TRUE;
   END_IF;
END_REGION

REGION Network 41: PFE Maintenance Faults 55
   RUNG wire#powerrail
      I_Contact( "Sensor".EM5[15] )
      { S7_Templates := "SrcType := LReal" } NE_Contact(in1 := "Unit1.Em5.ControlNodes".cmCathodeAlignTableAxisX.monitoring.actualPosition, in2 := 0.0)
      I_Contact( "Unit1.Em5.ControlNodes".cmCathodeAlignTableAxisX.monitoring.homingCommandBusy )
      { S7_Templates := "time_type := Time" } "Unit1.Em5.Alarms".tonMaintenanceFault[55].TON(pt := #DelayTime, et =>)
      Contact( false )
      S_Coil( "Unit1.Em5.Alarms".maintenanceFaults[55] )
   END_RUNG
   // the same network as SCL:
   "Unit1.Em5.Alarms".tonMaintenanceFault[55].TON(IN := NOT "Sensor".EM5[15] AND ("Unit1.Em5.ControlNodes".cmCathodeAlignTableAxisX.monitoring.actualPosition <> 0.0) AND NOT "Unit1.Em5.ControlNodes".cmCathodeAlignTableAxisX.monitoring.homingCommandBusy,
                           PT := #DelayTime);
   IF "Unit1.Em5.Alarms".tonMaintenanceFault[55].Q AND false THEN
       "Unit1.Em5.Alarms".maintenanceFaults[55] := TRUE;
   END_IF;
END_REGION

REGION Network 42: PFE Maintenance Faults 56
   RUNG wire#powerrail
      I_Contact( "Sensor".EM5[17] )
      { S7_Templates := "SrcType := LReal" } NE_Contact(in1 := "Unit1.Em5.ControlNodes".cmCathodeAlignTableAxisY1.monitoring.actualPosition, in2 := 0.0)
      I_Contact( "Unit1.Em5.ControlNodes".cmCathodeAlignTableAxisY1.monitoring.homingCommandBusy )
      { S7_Templates := "time_type := Time" } "Unit1.Em5.Alarms".tonMaintenanceFault[56].TON(pt := #DelayTime, et =>)
      Contact( false )
      S_Coil( "Unit1.Em5.Alarms".maintenanceFaults[56] )
   END_RUNG
   // the same network as SCL:
   "Unit1.Em5.Alarms".tonMaintenanceFault[56].TON(IN := NOT "Sensor".EM5[17] AND ("Unit1.Em5.ControlNodes".cmCathodeAlignTableAxisY1.monitoring.actualPosition <> 0.0) AND NOT "Unit1.Em5.ControlNodes".cmCathodeAlignTableAxisY1.monitoring.homingCommandBusy,
                           PT := #DelayTime);
   IF "Unit1.Em5.Alarms".tonMaintenanceFault[56].Q AND false THEN
       "Unit1.Em5.Alarms".maintenanceFaults[56] := TRUE;
   END_IF;
END_REGION

REGION Network 43: PFE Maintenance Faults 57
   RUNG wire#powerrail
      I_Contact( "Sensor".EM5[16] )
      { S7_Templates := "SrcType := LReal" } NE_Contact(in1 := "Unit1.Em5.ControlNodes".cmCathodeAlignTableAxisY2.monitoring.actualPosition, in2 := 0.0)
      I_Contact( "Unit1.Em5.ControlNodes".cmCathodeAlignTableAxisY2.monitoring.homingCommandBusy )
      { S7_Templates := "time_type := Time" } "Unit1.Em5.Alarms".tonMaintenanceFault[57].TON(pt := #DelayTime, et =>)
      Contact( false )
      S_Coil( "Unit1.Em5.Alarms".maintenanceFaults[57] )
   END_RUNG
   // the same network as SCL:
   "Unit1.Em5.Alarms".tonMaintenanceFault[57].TON(IN := NOT "Sensor".EM5[16] AND ("Unit1.Em5.ControlNodes".cmCathodeAlignTableAxisY2.monitoring.actualPosition <> 0.0) AND NOT "Unit1.Em5.ControlNodes".cmCathodeAlignTableAxisY2.monitoring.homingCommandBusy,
                           PT := #DelayTime);
   IF "Unit1.Em5.Alarms".tonMaintenanceFault[57].Q AND false THEN
       "Unit1.Em5.Alarms".maintenanceFaults[57] := TRUE;
   END_IF;
END_REGION

REGION Network 44: PFE Production Faults 0
   RUNG wire#powerrail
      Contact( false )
      { S7_Templates := "time_type := Time" } "Unit1.Em5.Alarms".tonProductionFault[0].TON(pt := #DelayTime, et =>)
      S_Coil( "Unit1.Em5.Alarms".productionFaults[0] )
   END_RUNG
   // the same network as SCL:
   "Unit1.Em5.Alarms".tonProductionFault[0].TON(IN := false, PT := #DelayTime);
   IF "Unit1.Em5.Alarms".tonProductionFault[0].Q THEN "Unit1.Em5.Alarms".productionFaults[0] := TRUE; END_IF;
END_REGION

REGION Network 45: PFE Production Faults 1
   RUNG wire#powerrail
      Contact( FALSE )
      S_Coil( "Unit1.Em5.Alarms".productionFaults[1] )
   END_RUNG
   // the same network as SCL:
   IF FALSE THEN "Unit1.Em5.Alarms".productionFaults[1] := TRUE; END_IF;
END_REGION

REGION Network 46: PFE Production Faults 2
   RUNG wire#powerrail
      Contact( FALSE )
      S_Coil( "Unit1.Em5.Alarms".productionFaults[2] )
   END_RUNG
   // the same network as SCL:
   IF FALSE THEN "Unit1.Em5.Alarms".productionFaults[2] := TRUE; END_IF;
END_REGION

REGION Network 47: PFE Production Faults 3
   RUNG wire#powerrail
      Contact( FALSE )
      S_Coil( "Unit1.Em5.Alarms".productionFaults[3] )
   END_RUNG
   // the same network as SCL:
   IF FALSE THEN "Unit1.Em5.Alarms".productionFaults[3] := TRUE; END_IF;
END_REGION

REGION Network 48: PFE Production Faults 4
   RUNG wire#powerrail
      Contact( FALSE )
      S_Coil( "Unit1.Em5.Alarms".productionFaults[4] )
   END_RUNG
   // the same network as SCL:
   IF FALSE THEN "Unit1.Em5.Alarms".productionFaults[4] := TRUE; END_IF;
END_REGION

REGION Network 49: PFE Tooling Faults 0
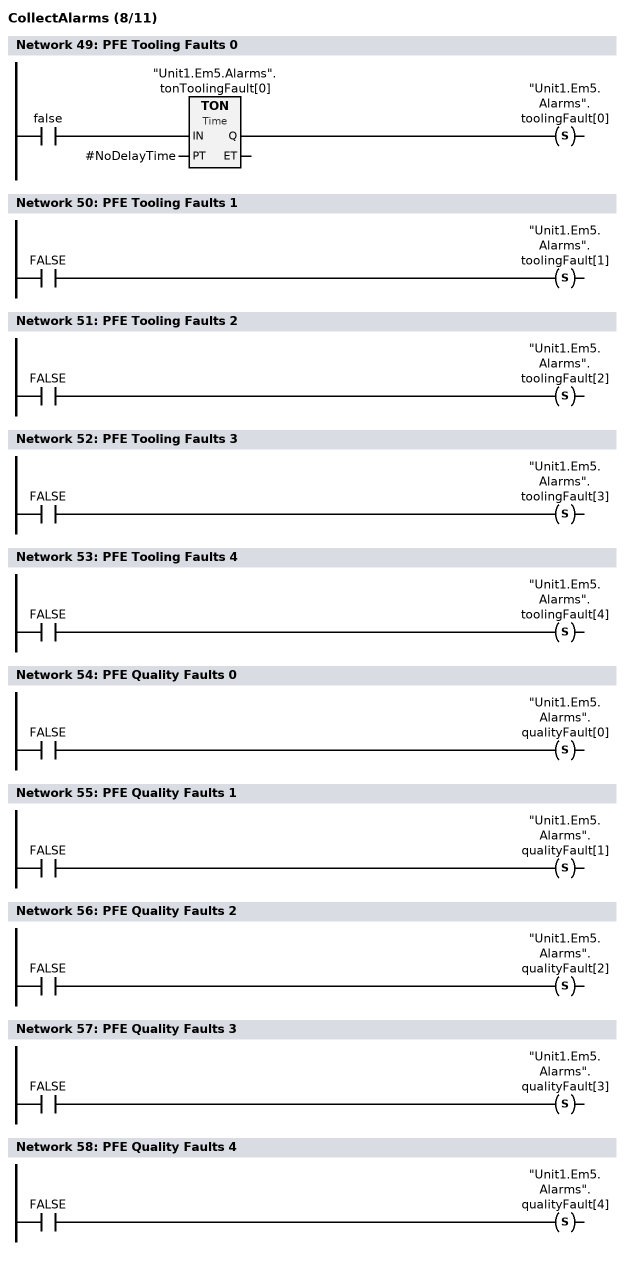
   RUNG wire#powerrail
      Contact( false )
      { S7_Templates := "time_type := Time" } "Unit1.Em5.Alarms".tonToolingFault[0].TON(pt := #NoDelayTime, et =>)
      S_Coil( "Unit1.Em5.Alarms".toolingFault[0] )
   END_RUNG
   // the same network as SCL:
   "Unit1.Em5.Alarms".tonToolingFault[0].TON(IN := false, PT := #NoDelayTime);
   IF "Unit1.Em5.Alarms".tonToolingFault[0].Q THEN "Unit1.Em5.Alarms".toolingFault[0] := TRUE; END_IF;
END_REGION

REGION Network 50: PFE Tooling Faults 1
   RUNG wire#powerrail
      Contact( FALSE )
      S_Coil( "Unit1.Em5.Alarms".toolingFault[1] )
   END_RUNG
   // the same network as SCL:
   IF FALSE THEN "Unit1.Em5.Alarms".toolingFault[1] := TRUE; END_IF;
END_REGION

REGION Network 51: PFE Tooling Faults 2
   RUNG wire#powerrail
      Contact( FALSE )
      S_Coil( "Unit1.Em5.Alarms".toolingFault[2] )
   END_RUNG
   // the same network as SCL:
   IF FALSE THEN "Unit1.Em5.Alarms".toolingFault[2] := TRUE; END_IF;
END_REGION

REGION Network 52: PFE Tooling Faults 3
   RUNG wire#powerrail
      Contact( FALSE )
      S_Coil( "Unit1.Em5.Alarms".toolingFault[3] )
   END_RUNG
   // the same network as SCL:
   IF FALSE THEN "Unit1.Em5.Alarms".toolingFault[3] := TRUE; END_IF;
END_REGION

REGION Network 53: PFE Tooling Faults 4
   RUNG wire#powerrail
      Contact( FALSE )
      S_Coil( "Unit1.Em5.Alarms".toolingFault[4] )
   END_RUNG
   // the same network as SCL:
   IF FALSE THEN "Unit1.Em5.Alarms".toolingFault[4] := TRUE; END_IF;
END_REGION

REGION Network 54: PFE Quality Faults 0
   RUNG wire#powerrail
      Contact( FALSE )
      S_Coil( "Unit1.Em5.Alarms".qualityFault[0] )
   END_RUNG
   // the same network as SCL:
   IF FALSE THEN "Unit1.Em5.Alarms".qualityFault[0] := TRUE; END_IF;
END_REGION

REGION Network 55: PFE Quality Faults 1
   RUNG wire#powerrail
      Contact( FALSE )
      S_Coil( "Unit1.Em5.Alarms".qualityFault[1] )
   END_RUNG
   // the same network as SCL:
   IF FALSE THEN "Unit1.Em5.Alarms".qualityFault[1] := TRUE; END_IF;
END_REGION

REGION Network 56: PFE Quality Faults 2
   RUNG wire#powerrail
      Contact( FALSE )
      S_Coil( "Unit1.Em5.Alarms".qualityFault[2] )
   END_RUNG
   // the same network as SCL:
   IF FALSE THEN "Unit1.Em5.Alarms".qualityFault[2] := TRUE; END_IF;
END_REGION

REGION Network 57: PFE Quality Faults 3
   RUNG wire#powerrail
      Contact( FALSE )
      S_Coil( "Unit1.Em5.Alarms".qualityFault[3] )
   END_RUNG
   // the same network as SCL:
   IF FALSE THEN "Unit1.Em5.Alarms".qualityFault[3] := TRUE; END_IF;
END_REGION

REGION Network 58: PFE Quality Faults 4
   RUNG wire#powerrail
      Contact( FALSE )
      S_Coil( "Unit1.Em5.Alarms".qualityFault[4] )
   END_RUNG
   // the same network as SCL:
   IF FALSE THEN "Unit1.Em5.Alarms".qualityFault[4] := TRUE; END_IF;
END_REGION

REGION Network 59: PFE Throughput Fault Blocked 0
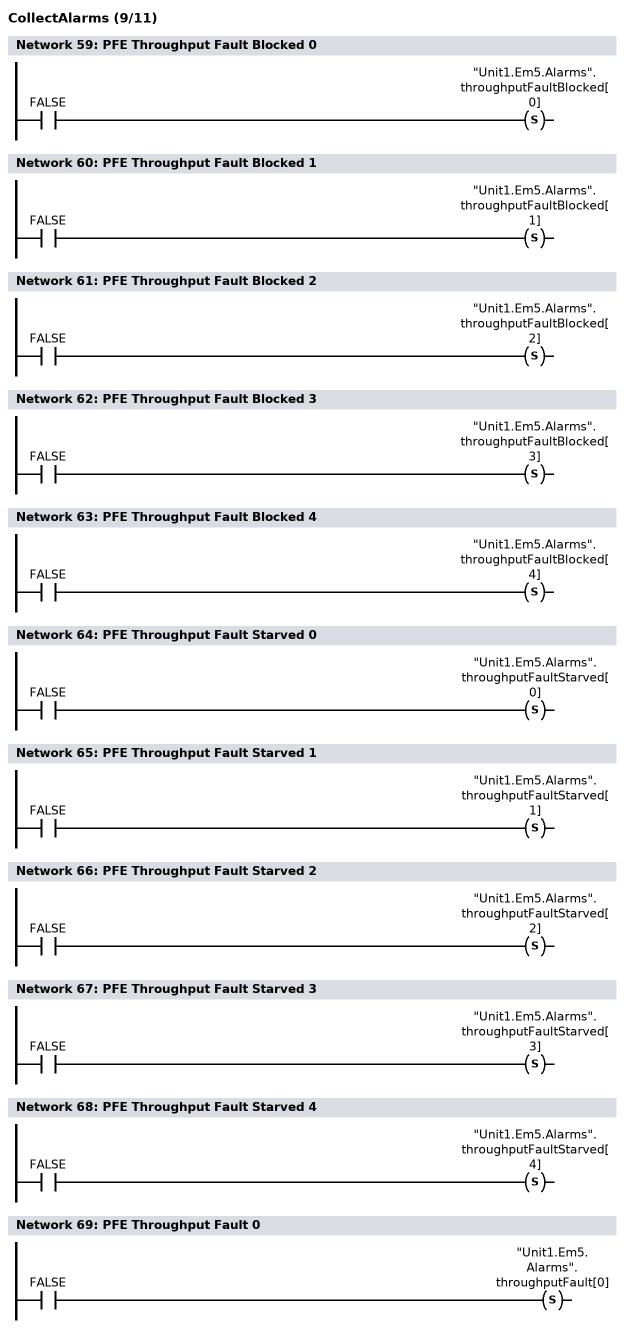
   RUNG wire#powerrail
      Contact( FALSE )
      S_Coil( "Unit1.Em5.Alarms".throughputFaultBlocked[0] )
   END_RUNG
   // the same network as SCL:
   IF FALSE THEN "Unit1.Em5.Alarms".throughputFaultBlocked[0] := TRUE; END_IF;
END_REGION

REGION Network 60: PFE Throughput Fault Blocked 1
   RUNG wire#powerrail
      Contact( FALSE )
      S_Coil( "Unit1.Em5.Alarms".throughputFaultBlocked[1] )
   END_RUNG
   // the same network as SCL:
   IF FALSE THEN "Unit1.Em5.Alarms".throughputFaultBlocked[1] := TRUE; END_IF;
END_REGION

REGION Network 61: PFE Throughput Fault Blocked 2
   RUNG wire#powerrail
      Contact( FALSE )
      S_Coil( "Unit1.Em5.Alarms".throughputFaultBlocked[2] )
   END_RUNG
   // the same network as SCL:
   IF FALSE THEN "Unit1.Em5.Alarms".throughputFaultBlocked[2] := TRUE; END_IF;
END_REGION

REGION Network 62: PFE Throughput Fault Blocked 3
   RUNG wire#powerrail
      Contact( FALSE )
      S_Coil( "Unit1.Em5.Alarms".throughputFaultBlocked[3] )
   END_RUNG
   // the same network as SCL:
   IF FALSE THEN "Unit1.Em5.Alarms".throughputFaultBlocked[3] := TRUE; END_IF;
END_REGION

REGION Network 63: PFE Throughput Fault Blocked 4
   RUNG wire#powerrail
      Contact( FALSE )
      S_Coil( "Unit1.Em5.Alarms".throughputFaultBlocked[4] )
   END_RUNG
   // the same network as SCL:
   IF FALSE THEN "Unit1.Em5.Alarms".throughputFaultBlocked[4] := TRUE; END_IF;
END_REGION

REGION Network 64: PFE Throughput Fault Starved 0
   RUNG wire#powerrail
      Contact( FALSE )
      S_Coil( "Unit1.Em5.Alarms".throughputFaultStarved[0] )
   END_RUNG
   // the same network as SCL:
   IF FALSE THEN "Unit1.Em5.Alarms".throughputFaultStarved[0] := TRUE; END_IF;
END_REGION

REGION Network 65: PFE Throughput Fault Starved 1
   RUNG wire#powerrail
      Contact( FALSE )
      S_Coil( "Unit1.Em5.Alarms".throughputFaultStarved[1] )
   END_RUNG
   // the same network as SCL:
   IF FALSE THEN "Unit1.Em5.Alarms".throughputFaultStarved[1] := TRUE; END_IF;
END_REGION

REGION Network 66: PFE Throughput Fault Starved 2
   RUNG wire#powerrail
      Contact( FALSE )
      S_Coil( "Unit1.Em5.Alarms".throughputFaultStarved[2] )
   END_RUNG
   // the same network as SCL:
   IF FALSE THEN "Unit1.Em5.Alarms".throughputFaultStarved[2] := TRUE; END_IF;
END_REGION

REGION Network 67: PFE Throughput Fault Starved 3
   RUNG wire#powerrail
      Contact( FALSE )
      S_Coil( "Unit1.Em5.Alarms".throughputFaultStarved[3] )
   END_RUNG
   // the same network as SCL:
   IF FALSE THEN "Unit1.Em5.Alarms".throughputFaultStarved[3] := TRUE; END_IF;
END_REGION

REGION Network 68: PFE Throughput Fault Starved 4
   RUNG wire#powerrail
      Contact( FALSE )
      S_Coil( "Unit1.Em5.Alarms".throughputFaultStarved[4] )
   END_RUNG
   // the same network as SCL:
   IF FALSE THEN "Unit1.Em5.Alarms".throughputFaultStarved[4] := TRUE; END_IF;
END_REGION

REGION Network 69: PFE Throughput Fault 0
   RUNG wire#powerrail
      Contact( FALSE )
      S_Coil( "Unit1.Em5.Alarms".throughputFault[0] )
   END_RUNG
   // the same network as SCL:
   IF FALSE THEN "Unit1.Em5.Alarms".throughputFault[0] := TRUE; END_IF;
END_REGION

REGION Network 70: PFE Throughput Fault 1
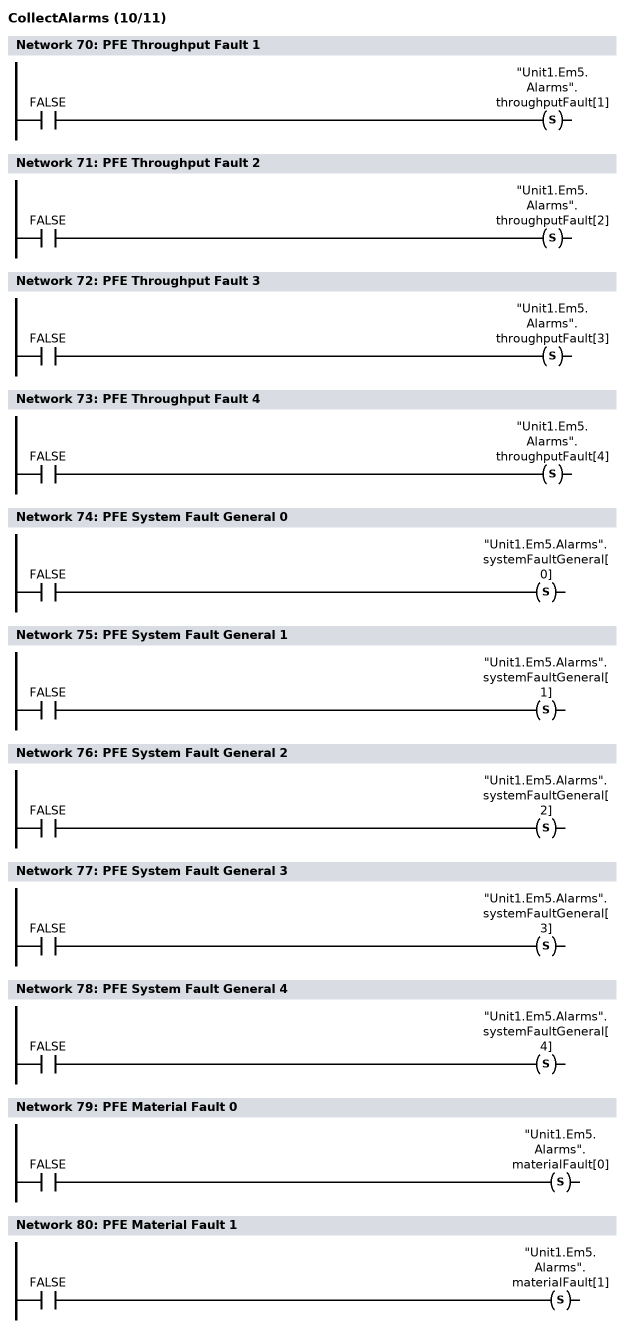
   RUNG wire#powerrail
      Contact( FALSE )
      S_Coil( "Unit1.Em5.Alarms".throughputFault[1] )
   END_RUNG
   // the same network as SCL:
   IF FALSE THEN "Unit1.Em5.Alarms".throughputFault[1] := TRUE; END_IF;
END_REGION

REGION Network 71: PFE Throughput Fault 2
   RUNG wire#powerrail
      Contact( FALSE )
      S_Coil( "Unit1.Em5.Alarms".throughputFault[2] )
   END_RUNG
   // the same network as SCL:
   IF FALSE THEN "Unit1.Em5.Alarms".throughputFault[2] := TRUE; END_IF;
END_REGION

REGION Network 72: PFE Throughput Fault 3
   RUNG wire#powerrail
      Contact( FALSE )
      S_Coil( "Unit1.Em5.Alarms".throughputFault[3] )
   END_RUNG
   // the same network as SCL:
   IF FALSE THEN "Unit1.Em5.Alarms".throughputFault[3] := TRUE; END_IF;
END_REGION

REGION Network 73: PFE Throughput Fault 4
   RUNG wire#powerrail
      Contact( FALSE )
      S_Coil( "Unit1.Em5.Alarms".throughputFault[4] )
   END_RUNG
   // the same network as SCL:
   IF FALSE THEN "Unit1.Em5.Alarms".throughputFault[4] := TRUE; END_IF;
END_REGION

REGION Network 74: PFE System Fault General 0
   RUNG wire#powerrail
      Contact( FALSE )
      S_Coil( "Unit1.Em5.Alarms".systemFaultGeneral[0] )
   END_RUNG
   // the same network as SCL:
   IF FALSE THEN "Unit1.Em5.Alarms".systemFaultGeneral[0] := TRUE; END_IF;
END_REGION

REGION Network 75: PFE System Fault General 1
   RUNG wire#powerrail
      Contact( FALSE )
      S_Coil( "Unit1.Em5.Alarms".systemFaultGeneral[1] )
   END_RUNG
   // the same network as SCL:
   IF FALSE THEN "Unit1.Em5.Alarms".systemFaultGeneral[1] := TRUE; END_IF;
END_REGION

REGION Network 76: PFE System Fault General 2
   RUNG wire#powerrail
      Contact( FALSE )
      S_Coil( "Unit1.Em5.Alarms".systemFaultGeneral[2] )
   END_RUNG
   // the same network as SCL:
   IF FALSE THEN "Unit1.Em5.Alarms".systemFaultGeneral[2] := TRUE; END_IF;
END_REGION

REGION Network 77: PFE System Fault General 3
   RUNG wire#powerrail
      Contact( FALSE )
      S_Coil( "Unit1.Em5.Alarms".systemFaultGeneral[3] )
   END_RUNG
   // the same network as SCL:
   IF FALSE THEN "Unit1.Em5.Alarms".systemFaultGeneral[3] := TRUE; END_IF;
END_REGION

REGION Network 78: PFE System Fault General 4
   RUNG wire#powerrail
      Contact( FALSE )
      S_Coil( "Unit1.Em5.Alarms".systemFaultGeneral[4] )
   END_RUNG
   // the same network as SCL:
   IF FALSE THEN "Unit1.Em5.Alarms".systemFaultGeneral[4] := TRUE; END_IF;
END_REGION

REGION Network 79: PFE Material Fault 0
   RUNG wire#powerrail
      Contact( FALSE )
      S_Coil( "Unit1.Em5.Alarms".materialFault[0] )
   END_RUNG
   // the same network as SCL:
   IF FALSE THEN "Unit1.Em5.Alarms".materialFault[0] := TRUE; END_IF;
END_REGION

REGION Network 80: PFE Material Fault 1
   RUNG wire#powerrail
      Contact( FALSE )
      S_Coil( "Unit1.Em5.Alarms".materialFault[1] )
   END_RUNG
   // the same network as SCL:
   IF FALSE THEN "Unit1.Em5.Alarms".materialFault[1] := TRUE; END_IF;
END_REGION

REGION Network 81: PFE Material Fault 2
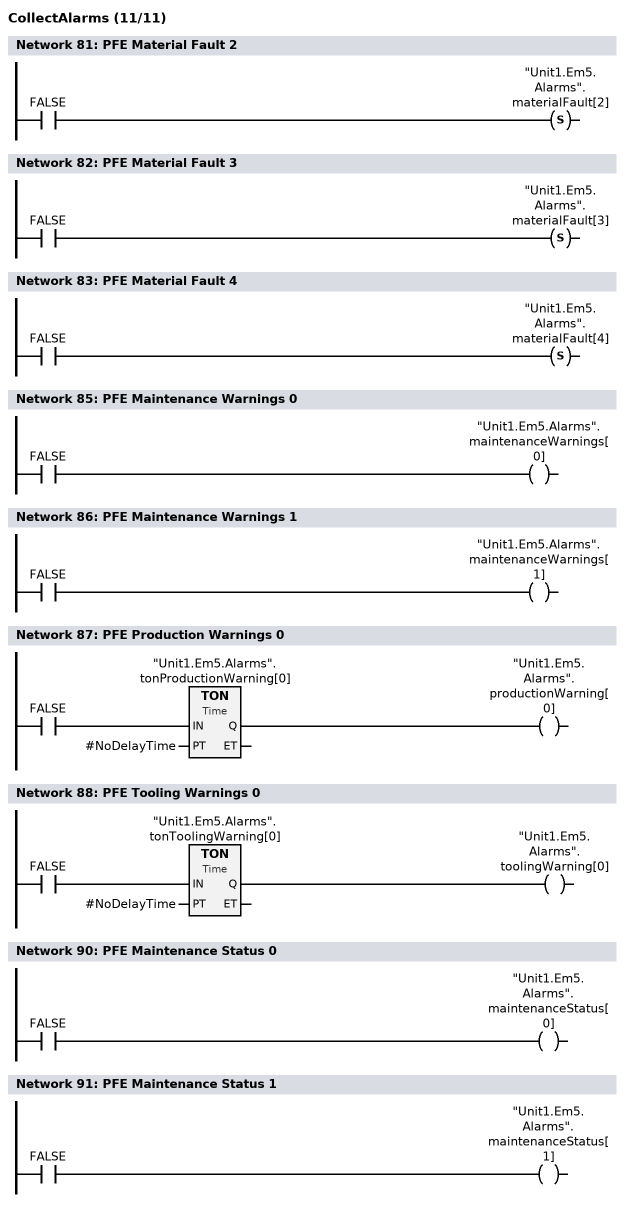
   RUNG wire#powerrail
      Contact( FALSE )
      S_Coil( "Unit1.Em5.Alarms".materialFault[2] )
   END_RUNG
   // the same network as SCL:
   IF FALSE THEN "Unit1.Em5.Alarms".materialFault[2] := TRUE; END_IF;
END_REGION

REGION Network 82: PFE Material Fault 3
   RUNG wire#powerrail
      Contact( FALSE )
      S_Coil( "Unit1.Em5.Alarms".materialFault[3] )
   END_RUNG
   // the same network as SCL:
   IF FALSE THEN "Unit1.Em5.Alarms".materialFault[3] := TRUE; END_IF;
END_REGION

REGION Network 83: PFE Material Fault 4
   RUNG wire#powerrail
      Contact( FALSE )
      S_Coil( "Unit1.Em5.Alarms".materialFault[4] )
   END_RUNG
   // the same network as SCL:
   IF FALSE THEN "Unit1.Em5.Alarms".materialFault[4] := TRUE; END_IF;
END_REGION

REGION Network 84: *************** Warning **************************
END_REGION

REGION Network 85: PFE Maintenance Warnings 0
   RUNG wire#powerrail
      Contact( FALSE )
      Coil( "Unit1.Em5.Alarms".maintenanceWarnings[0] )
   END_RUNG
   // the same network as SCL:
   "Unit1.Em5.Alarms".maintenanceWarnings[0] := FALSE;
END_REGION

REGION Network 86: PFE Maintenance Warnings 1
   RUNG wire#powerrail
      Contact( FALSE )
      Coil( "Unit1.Em5.Alarms".maintenanceWarnings[1] )
   END_RUNG
   // the same network as SCL:
   "Unit1.Em5.Alarms".maintenanceWarnings[1] := FALSE;
END_REGION

REGION Network 87: PFE Production Warnings 0
   RUNG wire#powerrail
      Contact( FALSE )
      { S7_Templates := "time_type := Time" } "Unit1.Em5.Alarms".tonProductionWarning[0].TON(pt := #NoDelayTime, et =>)
      Coil( "Unit1.Em5.Alarms".productionWarning[0] )
   END_RUNG
   // the same network as SCL:
   "Unit1.Em5.Alarms".tonProductionWarning[0].TON(IN := FALSE, PT := #NoDelayTime);
   "Unit1.Em5.Alarms".productionWarning[0] := "Unit1.Em5.Alarms".tonProductionWarning[0].Q;
END_REGION

REGION Network 88: PFE Tooling Warnings 0
   RUNG wire#powerrail
      Contact( FALSE )
      { S7_Templates := "time_type := Time" } "Unit1.Em5.Alarms".tonToolingWarning[0].TON(pt := #NoDelayTime, et =>)
      Coil( "Unit1.Em5.Alarms".toolingWarning[0] )
   END_RUNG
   // the same network as SCL:
   "Unit1.Em5.Alarms".tonToolingWarning[0].TON(IN := FALSE, PT := #NoDelayTime);
   "Unit1.Em5.Alarms".toolingWarning[0] := "Unit1.Em5.Alarms".tonToolingWarning[0].Q;
END_REGION

REGION Network 89: *************** Status ***************************
END_REGION

REGION Network 90: PFE Maintenance Status 0
   RUNG wire#powerrail
      Contact( FALSE )
      Coil( "Unit1.Em5.Alarms".maintenanceStatus[0] )
   END_RUNG
   // the same network as SCL:
   "Unit1.Em5.Alarms".maintenanceStatus[0] := FALSE;
END_REGION

REGION Network 91: PFE Maintenance Status 1
   RUNG wire#powerrail
      Contact( FALSE )
      Coil( "Unit1.Em5.Alarms".maintenanceStatus[1] )
   END_RUNG
   // the same network as SCL:
   "Unit1.Em5.Alarms".maintenanceStatus[1] := FALSE;
END_REGION
END_FUNCTION
